Staubli VAL3: onStart.pgx

public program onStart(string& x_sItem[])
// check and put all the boolean as the status of BIO-MIO-MODBUS-FIELDBUS-ARMIO
  local num i
  local num l_nModbusOut
  local num l_nFieldbusOut
  local bool l_bChange
  local num l_nResult
  local string l_sPath
  local bool l_bCheck
  local string l_sKey
begin
  if x_sItem=="init"
    //
    // DIGITAL INPUT
    //
    // set the default value
    call saveInOut:setOutput(0)
//    // BIO
//    call saveInOut:setOutput(1)
//    // BIO2 - MIO
//    call saveInOut:setOutput(2)
//    // MODBUS
//    call saveInOut:setOutput(3)
//    // USER
//    call saveInOut:setOutput(4)
//    // REMIO
    //    call saveInOut:setOutput(5)
    call saveInOut:setOutput(6)
    //
    // SAVE
    //
    call save(l_nResult)
    if l_nResult==0
      logMsg("[KERNEL] SUPERVISOR>Output: Save Done")
    else
      logMsg("error "+toString("",l_nResult)+" saving the saveInputOutput")
      popUpMsg("error "+toString("",l_nResult)+" saving the saveInputOutput")
    endIf
  endIf
  // build the list for easy access
  // start from the first
  resize(sKey,1,1)
  sKey=""
  if isDefined(saveInOut:dOutput["valve1"])
    sKey[0]="valve1"
  endIf
  if isDefined(saveInOut:dOutput["valve2"])
    append(sKey)
    sKey[1]="valve2"
  endIf
  if isDefined(saveInOut:dOutput["fOut0"])
    append(sKey)
    sKey[2]="fOut0"
  endIf
  l_sKey=first(saveInOut:dOutput)
  i=size(sKey)-1
  // search it
  //
  while l_sKey!=""
    if find(l_sKey,"valve")==-1 and find(l_sKey,"fOut")==-1
      if !(sKey[0]=="" and i==0)
        append(sKey)
        i=i+1
      endIf
      sKey[i]=l_sKey
    endIf
    l_sKey=next(saveInOut:dOutput[l_sKey])
  endWhile
end
